Staubli VAL3: getSize.pgx

public program getSize(num& x_nSize[] (dimensions=1))
begin
end
